FUNCTION_BLOCK FB_Homing_Mock EXTENDS FB_CyclicFB IMPLEMENTS I_MotionSequence
VAR
	// Wewnętrzne flagi interfejsu
    _bBusy    : BOOL;
    _bInitComplete    : BOOL;
	_bDone :BOOL;
    _bError   : BOOL;
    _iErrorID : UDINT;
    
    // Zmienne naszego Mocka
    nStep    : INT;
    tTimer   : TON;
    
    // Referencja do osi (żeby wymusić flagę Homed)
    _Axis    : I_BasicAxis;
    fbSetPos : MC_SetPosition;
END_VAR


PROPERTY Axis : SPT_Motion_Control.I_BasicAxis
GET
Axis := _Axis;
END_GET
SET
_Axis := Axis;
END_SET
END_PROPERTY

PROPERTY Busy : BOOL
GET
Busy:=_bBusy;
END_GET
END_PROPERTY

METHOD PUBLIC CyclicLogic
CASE nStep OF
    0:
        // Idle - czekamy na Execute
        
    10:
        // Udajemy bazowanie - czekamy 2 sekundy
        tTimer(IN := TRUE, PT := T#2S);
        
        IF tTimer.Q THEN
            tTimer(IN := FALSE);
            nStep := 20;
        END_IF
        
    20:
        // Oszukujemy NC - ustawiamy pozycję na 0.0 i wymuszamy flagę Homed
        fbSetPos(
            Axis     := _Axis.Axis, 
            Execute  := TRUE, 
            Position := 0.0, 
            Mode     := FALSE // Wymusza absolutne ustawienie pozycji
        );
        
        IF fbSetPos.Done THEN
            fbSetPos(Axis := _Axis.Axis, Execute := FALSE); // Reset bloku
            nStep := 30;
        END_IF
        
    30:
        // Sukces!
        _bBusy := FALSE;
        _bDone := TRUE;
        nStep := 0;
        
END_CASE
END_METHOD


PROPERTY Error : BOOL
GET
Error := _bError;
END_GET
END_PROPERTY


PROPERTY ErrorID : UDINT
GET
ErrorID := _iErrorID;
END_GET
END_PROPERTY

METHOD PUBLIC Execute : BOOL
IF nStep = 0 THEN
    _bBusy    := TRUE;
    _bDone    := FALSE;
    _bError   := FALSE;
    _iErrorID := 0;
    nStep    := 10;
END_IF

Execute := TRUE; // Potwierdzamy przyjęcie rozkazu
END_METHOD

PROPERTY InitComplete : BOOL
GET
InitComplete := _bInitComplete;
END_GET
END_PROPERTY

END_FUNCTION_BLOCK

(* stored: Version 1.1.0.1, ProductVersion 3.1.4024.15
   POU FB_Homing_Mock: Id {e31a3749-123b-4dfb-ad39-aa25645894ff}, SpecialFunc None
   Property Axis: Id {0f65bf00-67fe-4aba-8137-b51d116c1159}
   Get Get: Id {e9e4b2b8-db7b-4d3f-90bf-522581a11a2c}
   Set Set: Id {f6d5b25c-c61c-4423-b3ae-eca06aecc471}
   Property Busy: Id {43351339-3329-4098-9bdf-09b26ee270da}
   Get Get: Id {81eeacd2-966d-4849-b300-eeeb505be167}
   Method CyclicLogic: Id {17f462d7-3d9f-4c9b-bb5b-b5a89fe32605}
   Property Error: Id {833f06a6-c2fe-4eb5-9e4d-6e7b38e40001}
   Get Get: Id {0808e801-ef4f-4a63-99a7-98f653003203}
   Property ErrorID: Id {b89fed01-dea3-431d-b1bd-6f652b1e4c5f}
   Get Get: Id {9b26b192-a953-4eb3-bdfe-c36ba145afad}
   Method Execute: Id {938833ed-e6b3-4e5e-9c5c-e8e12ac7416a}
   Property InitComplete: Id {eb4b3d66-90ef-4785-803b-ec27b572a39e}
   Get Get: Id {fd92954a-0b4b-49ed-9012-202593124c18} *)
